// TwinCAT 3 PLC project PLC3
// ProgramVersion: 3.1.4022.3
// libraries:
//   Tc2_Standard, * (Beckhoff Automation GmbH)
//   Tc2_System, * (Beckhoff Automation GmbH)
//   Tc3_Module, * (Beckhoff Automation GmbH)
// project tree:
//   DUTs/ States.TcDUT
//   GVLs/ GVL_IO.TcGVL (not stored)
//   / PlcTask.TcTTO (not stored)
//   POUs/ MAIN.TcPOU

// ---- DUTs/States.TcDUT
{attribute 'qualified_only'}
{attribute 'strict'}
TYPE States :
(
	Init := 0,
	Idle,
	MoveToPickUp,
	PickUpDown,
	PickUpUp,
	MoveX,
	MoveY,
	DropDown,
	DropUp,
	PalletFull
);
END_TYPE

// ---- POUs/MAIN.TcPOU
PROGRAM MAIN
VAR

	Timer1 :TON;
	Timer2 : TON;
	PulseTimer1 : TP;
	PulseTimer2 : TP;

	CurrentState  : States;
	
	ServoRTrigY : R_Trig ; 
	ServoRTrigX : R_Trig ; 
	
	BusyFtrigX : F_Trig;
	BusyFtrigY : F_Trig;
	
	
	//Eigen trigger booleans
	InitYReady : BOOL;
	InitXReady : BOOL;
	
	ReadyX : BOOL;
	ReadyY : BOOL;
	
	Full : BOOL;
	Busy : BOOL;
	
END_VAR

PulseTimer1(IN:=GVL_IO.Start_button, PT:=T#150MS);
PulseTimer2(IN:=Busy, PT:=T#150MS);

Timer1(IN:= GVL_IO.a_1_Vertical_Zaxis_downward, PT:= T#10MS);

CASE CurrentState OF
States.Init:
		//Aanzetten van servo's. Dit kan even duren GEEN HOMING
		GVL_IO.SVONX_SERVO_ON_tableX 	  := TRUE; 
		GVL_IO.SVONY_SERVO_ON_translY 	  := TRUE;
		
		GVL_IO.SETUPX_ORIGIN_tableX := PulseTimer1.Q;
		GVL_IO.SETUPY_ORIGIN_translY := PulseTimer1.Q;
		
		//// Koppelen van outputs Busy aan var's. Triggered op een falling edge.
		IF PulseTimer1.Q THEN
			ServoRTrigX ( clk := gvl_io.SETONX_ORIGIN_tableX ); 
	  		ServoRTrigY ( clk := gvl_io.SETONY_ORIGIN_translationY );
		END_IF
		
		// Bools setten aan de hand van triggers.
		IF ServoRTrigX.Q THEN
			InitXReady:= TRUE;
		END_IF
		
		IF ServoRTrigY.Q THEN
			InitYReady:= TRUE;
		END_IF
		
		// Init voltooid ga naar idle
		IF InitXReady AND InitYReady THEN
			CurrentState:= States.Idle;
		END_IF
		
States.Idle:
		IF NOT GVL_IO.Stop_button AND NOT GVL_IO.dp2_Cover_detection THEN
			//SEND MESSAGEE TODO
			CurrentState := States.Idle;
		END_IF
		
		IF NOT GVL_IO.Stop_button AND GVL_IO.dp1_Can_detection AND GVL_IO.dp2_Cover_detection AND NOT Full THEN
			CurrentState := States.MoveToPickUp; //TODO stopbutton
		END_IF
		
		IF Full THEN
			CurrentState := States.PalletFull;
		END_IF
		
States.MoveToPickUp:
		Busy := TRUE;
		GVL_IO.INX0_from_Input0_tableX := FALSE;
		GVL_IO.INX1_from_Input1_tableX := FALSE;
		GVL_IO.INX2_from_Input2_tableX := TRUE;
		GVL_IO.INY0_from_Input0_translY := TRUE;
		GVL_IO.INY1_from_Input1_translY := FALSE;
		GVL_IO.INY2_from_Input2_translY := TRUE;
		GVL_IO.DRIVEX_MOVE_tableX := PulseTimer2.Q;
		GVL_IO.DRIVEY_MOVE_translY := PulseTimer2.Q;
		
		//// Koppelen van outputs Busy aan var's. Triggered op een falling edge.
	   	BusyFtrigX ( clk := gvl_io.BUSYX_BUSY_tableX ); 
	  	BusyFtrigY ( clk := gvl_io.BUSYY_BUSY_traslationY );
		
		// Bools setten aan de hand van triggers.
		IF BusyFtrigX.Q THEN
			ReadyX:= TRUE;
		END_IF
		
		IF BusyFtrigY.Q THEN
			ReadyY:= TRUE;
		END_IF
		
		// Init voltooid ga naar idle
		IF ReadyY AND ReadyX THEN
			GVL_IO.DRIVEX_MOVE_tableX := FALSE;
			GVL_IO.DRIVEY_MOVE_translY := FALSE;
			ReadyX:= FALSE;
			ReadyY:= FALSE;
			Busy:= FALSE;
			CurrentState := States.PickUpDown;
		END_IF
		
States.PickUpDown:
		IF GVL_IO.a_0_Vertical_Zaxis_upward THEN
			GVL_IO.Aplus_Vert_axis_downwards := TRUE;
		END_IF
		
		IF GVL_IO.a_1_Vertical_Zaxis_downward THEN
			GVL_IO.Vplus_Vacuum_start := TRUE;
			
			IF Timer1.Q THEN
			CurrentState := States.PickUpUp;
			END_IF
		END_IF

States.PickUpUp:
		GVL_IO.Aplus_Vert_axis_downwards := FALSE;
		
		IF GVL_IO.a_0_Vertical_Zaxis_upward THEN
			CurrentState := States.MoveX;
		END_IF
		
States.MoveX:
		CurrentState := States.MoveY;
		
States.MoveY:
		CurrentState := States.DropDown;
		
States.DropDown:
		IF GVL_IO.a_0_Vertical_Zaxis_upward THEN
			GVL_IO.Aplus_Vert_axis_downwards := TRUE;
		END_IF
		
		IF 	GVL_IO.a_1_Vertical_Zaxis_downward THEN
			GVL_IO.Vplus_Vacuum_start := FALSE;
			Timer2(IN:=GVL_IO.a_1_Vertical_Zaxis_downward, PT:=T#10MS);
			IF Timer2.Q THEN
				CurrentState := States.DropUp;
			END_IF
		END_IF


States.DropUp:
		IF GVL_IO.a_1_Vertical_Zaxis_downward THEN
			GVL_IO.Aplus_Vert_axis_downwards := FALSE;
		END_IF
		
		IF GVL_IO.a_0_Vertical_Zaxis_upward THEN
			CurrentState := States.Idle;
		END_IF
END_CASE

END_PROGRAM
